// Mitsubishi GX Works2 project: LRI - PLC - NAND   PLC: Q03UDV

PROGRAM MAIN
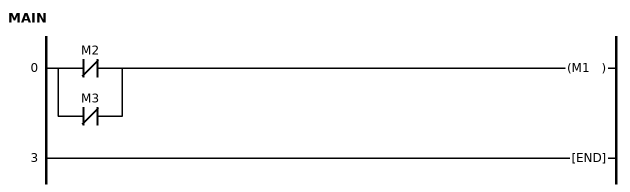
0     LDI     M2
      ORI     M3
      OUT     M1
3     END
END_PROGRAM
